PROGRAM MAIN
VAR
END_VAR

END_PROGRAM

(* stored: Version 1.1.0.1
   POU MAIN: Id {00a6aee8-9399-413c-9503-e45913b5af8b} *)
